FUNCTION_BLOCK COLOR_DECIDER (* Basic Function Block Type *)
  (* Standard: 61499-2 *)
  (* Version 0.3, 2009-09-15, JHC, Holobloc Inc, Changed transition priorities. *)
  (* Version 0.2, 2003-12-04, JHC, Rockwell Automation, Renamed for better indexing. *)
  (* Version 0.1, 2002-11-05, JHC, Rockwell Automation, Corrected missing ST element in Algorithm REQ. *)
  (* Version 0.0, 2000-05-30, JHC, Rockwell Automation *)
  PACKAGE fb.rt.Conveyer;
  IMPORT fb.datatype.*;
  IMPORT fb.rt.*;
  IMPORT fb.rt.mva.VSTYLE;
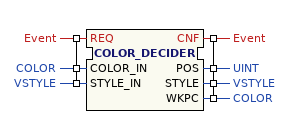
  EVENT_INPUT
    REQ WITH COLOR_IN, STYLE_IN;
  END_EVENT
  EVENT_OUTPUT
    CNF WITH POS, STYLE, WKPC; (* Execution Confirmation *)
  END_EVENT
  VAR_INPUT
    COLOR_IN : COLOR;
    STYLE_IN : VSTYLE;
  END_VAR
  VAR_OUTPUT
    POS : UINT := 0;
    STYLE : VSTYLE := PALLET;
    WKPC : COLOR;
  END_VAR
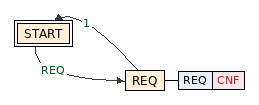
  EC_STATES
    START; (* Initial State *)
    REQ : REQ -> CNF;
  END_STATES
  EC_TRANSITIONS
    START TO REQ := REQ;
    REQ TO START := 1;
  END_TRANSITIONS
  ALGORITHM REQ IN ST:
POS := 0;
STYLE := STYLE_IN;
WKPC := COLOR_IN;
  END_ALGORITHM
END_FUNCTION_BLOCK
